ABB RobotStudio station: Project1.rsstnx

Station Project1 (saved by RobotStudio 25.2.11266.1)
Controller Controller1
  mechanical unit ROB_1: IRB140_6_81_C_03, 6 joints, base frame (0, 0, 0) mm
Layout (positions relative to the parent item):
  - IRB140_6_81_C_03 [mechanism, from %ABB.RobotStudio.Models.IRB140%\IRB140_6_81_C_G_03.rslib] at (0, 0, 0) mm; joint values [0, 0, 0, 0, 0.5236, 0] (rad or m)
  - MyTool [mechanism, from Training Objects\myTool.rslib] at (506.29, 0, 679.5) mm, rotated rx 180 ry 60 rz 180 deg
  - table_and_fixture_140 [part, from Training Objects\propeller_table.rslib] at (800, -225, 0) mm, rotated rx 0 ry 0 rz 90 deg
Attachment: MyTool is attached to IRB140_6_81_C_03 / Link6
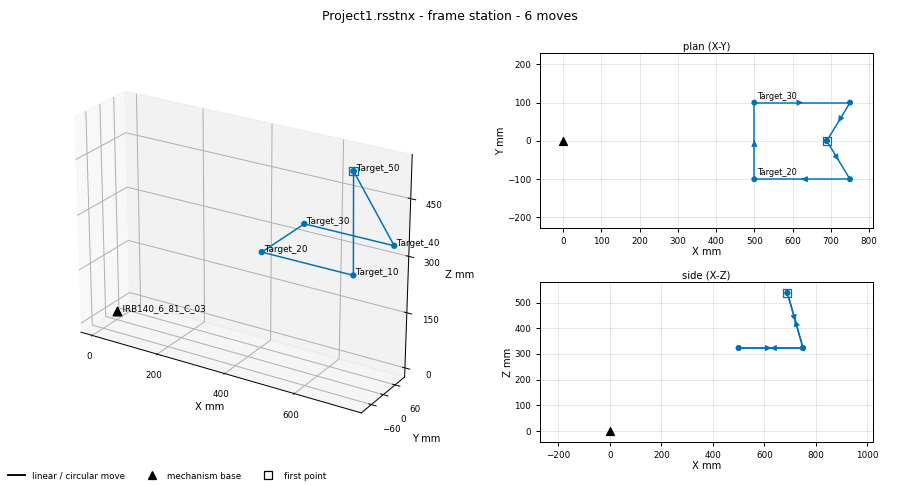
[picture p0: tool path of Project1.rsstnx in frame station, 6 of 6 moves have a stored position in this frame; points joined in program order, loops and branches not executed]
Targets, tools, work objects and paths stored in the station, written as RAPID:
! task T_ROB1
MODULE CalibData
  PERS tooldata MyTool:=[TRUE,[[31.792631019,0,229.638935148],[0.945518576,0,0.325568154,0]],[1,[0,0,1],[1,0,0,0],0,0,0]];
  TASK PERS wobjdata Workobject_1:=[FALSE,TRUE,"",[[475,-199.049,308],[0,0.707106781,0.707106781,0]],[[0,0,0],[1,0,0,0]]];
ENDMODULE

! task T_ROB1
MODULE Module1
  CONST robtarget Target_10:=[[99.049,275,-15],[0.707106781,0,0,-0.707106781],[0,0,0,0],[9E+09,9E+09,9E+09,9E+09,9E+09,9E+09]];
  CONST robtarget Target_20:=[[99.049,25,-15],[0.707106781,0,0,-0.707106781],[-1,0,-1,0],[9E+09,9E+09,9E+09,9E+09,9E+09,9E+09]];
  CONST robtarget Target_30:=[[299.049,25,-15],[0.707106781,0,0,-0.707106781],[0,-1,0,0],[9E+09,9E+09,9E+09,9E+09,9E+09,9E+09]];
  CONST robtarget Target_40:=[[299.049,275,-15],[0.707106781,0,0,-0.707106781],[0,-1,0,0],[9E+09,9E+09,9E+09,9E+09,9E+09,9E+09]];
  CONST robtarget Target_50:=[[199.049,214.268487273,-229.14730631],[0.694115238,-0.134922335,-0.134922335,-0.694115238],[0,0,0,0],[9E+09,9E+09,9E+09,9E+09,9E+09,9E+09]];
  PROC Path_10()
    MoveL Target_50,v300,fine,MyTool\WObj:=Workobject_1;
    MoveL Target_10,v300,fine,MyTool\WObj:=Workobject_1;
    MoveL Target_20,v300,fine,MyTool\WObj:=Workobject_1;
    MoveL Target_30,v300,fine,MyTool\WObj:=Workobject_1;
    MoveL Target_40,v300,fine,MyTool\WObj:=Workobject_1;
    MoveL Target_50,v300,fine,MyTool\WObj:=Workobject_1;
  ENDPROC
ENDMODULE

